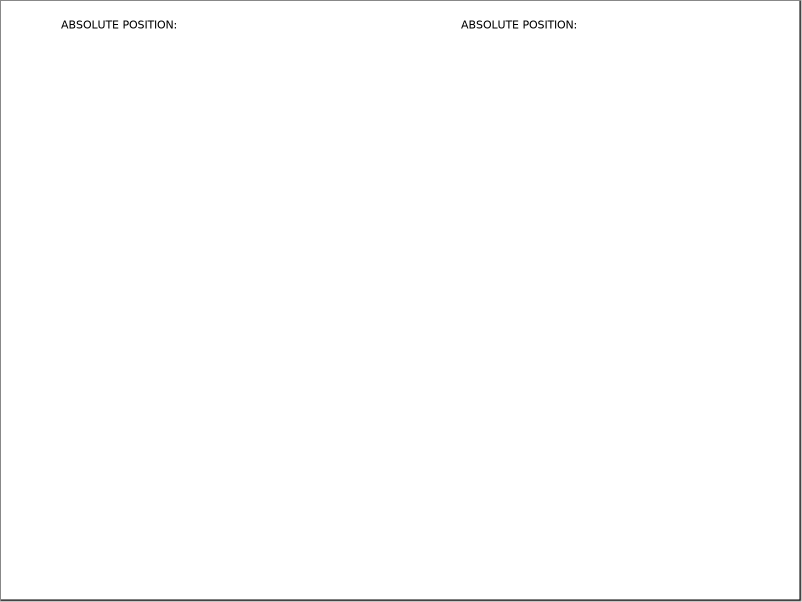
VISUALIZATION F10_Read_Digital_Output  // 802x602
    Rectangle (0,0 800x600)
    Label (10,10 170x30), "ABSOLUTE POSITION:"
    Label (410,10 170x30), "ABSOLUTE POSITION:"
END_VISUALIZATION

(* stored: Version 1.1.0.1, ProductVersion 3.1.4022.7
   Visu F10_Read_Digital_Output: Id {22af2caa-227d-4217-b487-059fb71f6dd2} *)
